// TwinCAT 3 PLC project Hboy
// ProgramVersion: 3.1.4023.0
// libraries:
//   Tc2_MC2, * (Beckhoff Automation GmbH)
//   Tc2_Standard, * (Beckhoff Automation GmbH)
//   Tc2_System, * (Beckhoff Automation GmbH)
//   Tc2_SystemCX, * (Beckhoff Automation GmbH)
//   Tc2_Utilities, * (Beckhoff Automation GmbH)
//   Tc3_Module, * (Beckhoff Automation GmbH)
//   XboxControllerUtilities, * (Beckhoff Community)
// project tree:
//   DUTs/ Controller.TcDUT, Pos.TcDUT
//   GVLs/ GVL.TcGVL
//   / PlcTask.TcTTO
//   POUs/ E_Stop.TcPOU, HbotForwardKinematics.TcPOU, LimitSwitches.TcPOU, TcXbox.TcPOU, MovementTypeSelector.TcPOU, PrepareAxes.TcPOU, MAIN.TcPOU
//   POUs/MovementType_Gcode/ FB_Movement_Gcode.TcPOU, FB_GcodeAgent.TcPOU
//   POUs/MovementType_Teach/ FB_Frames.TcPOU, FB_Movement_Teach.TcPOU, FB_Movement_Xbox.TcPOU, Frame.TcDUT
//   POUs/Hbot_Kinematics/ FB_HbotHome.TcPOU, FB_HbotKinematics.TcPOU, FB_HbotMovement.TcPOU, FB_PowerAll.TcPOU, FB_ResetAll.TcPOU
// real-time tasks:
//   TASK PlcTask: cycle T#1ms, priority 20, ADS port 350
//   TASK Job Task: cycle default, priority 32
// motion (NC):
//   TASK NC-Task 1 SAF: cycle T#2ms, priority 4, ADS port 501
//   TASK NC-Task 1 SVB: cycle T#10ms, priority 8, ADS port 511
//   AXIS Axis A (id 1)
//     Dynamic: Acceleration=20631.2, Deceleration=20631.2, Jerk=1237870, DelayTime=0.008
//     Velo: RefSearch=6.87706, RefSync=6.87706, SlowManual=150, FastManual=200, Fast=2347.941, Maximum=687.706
//     OtherSettings: AllowMotionCmdToSlave=true
//     encoder EncType=19
//       EncPara: ScaleFactorNumerator=60, ScaleFactorDenominator=1048576, MaxCount=#xffffffff
//     drive DrvType=16
//       DrvPara: MaxCount=#xffffffff, DriveControlDWord=#x00020100
//         Analog: VeloReferenz=756.4766, TorqueSetpointScale=10, ScaleFactorActTorque=0.1
//         TimeComp: TaskDelayCycles=1
//     controller CtrType=1
//       CtrPara: PriorControlFactor=1
//         PosDiffControl: Enable=false
//         Observer: BandWidth=20
//   AXIS Axis B (id 2)
//     Dynamic: Acceleration=15768.4, Deceleration=15768.4, Jerk=2468790, DelayTime=0.008
//     Velo: RefSearch=6.87706, RefSync=6.87706, SlowManual=150, FastManual=200, Fast=687.706, Maximum=687.706
//     OtherSettings: AllowMotionCmdToSlave=true
//     encoder EncType=19
//       EncPara: ScaleFactorNumerator=60, ScaleFactorDenominator=1048576, Inverse=true, MaxCount=#xffffffff
//     drive DrvType=16
//       DrvPara: Inverse=true, MaxCount=#xffffffff, DriveControlDWord=#x00020100
//         Analog: VeloReferenz=756.4766, TorqueSetpointScale=10, ScaleFactorActTorque=0.1
//         TimeComp: TaskDelayCycles=1
//     controller CtrType=1
//       CtrPara: PriorControlFactor=1
//         PosDiffControl: Enable=false
//         Observer: BandWidth=20
// I/O:
//   DEVICE Device 1 (EtherCAT), AmsNetId 5.71.241.84.2.1
//     Term 1 (EK1200) [EK1200-5000 EtherCAT Power supply (2A E-Bus)]
//       Term 8 (EL1012) [EL1012 2Ch. Dig. Input 24V, 10µs]
//       Term 2 (EL6900) [EL6900, TwinSAFE PLC]
//       Term 3 (EL1904) [EL1904, 4 Ch. Safety Input 24V, TwinSAFE]
//         modules: Module 1 (FSOES)
//       Term 4 (EL2904) [EL2904, 4 Ch. Safety Output 24V, 0.5A, TwinSAFE]
//         modules: Module 1 (FSOES), Module 2 (DO)
//       Term 5 (ELM7222-0010) [ELM7222-0010 2Ch. Servo Terminal (48 V, 8 A RMS, OCT)]
//       Term 6 (EL1088) [EL1088 8Ch. Dig. Input 24V, 3ms, negative]
//       Term 7 (EL9011) [EL9011 End Terminal]
//   DEVICE Device 5 (USB)
//     Box 1 (CX2100 Power Supply)
// variable links:
//   Device 1 (EtherCAT) <-> Device 1 (EtherCAT)/Term 1 (EK1200)/Term 2 (EL6900)
//     Term 1 (EK1200)/Term 3 (EL1904)/Module 1 (FSOES)/RxPDO/FSOE <-> ConnectionInputs/Message_9 TxPDO
//     Term 1 (EK1200)/Term 4 (EL2904)/Module 1 (FSOES)/RxPDO/FSOE <-> ConnectionInputs/Message_10 TxPDO
//     Term 1 (EK1200)/Term 3 (EL1904)/Module 1 (FSOES)/TxPDO/FSOE <-> ConnectionOutputs/Message_9 RxPDO
//   Device 1 (EtherCAT) <-> Device 1 (EtherCAT)/Term 1 (EK1200)/Term 4 (EL2904)
//     Term 1 (EK1200)/Term 2 (EL6900)/ConnectionOutputs/Message_10 RxPDO <-> Module 1 (FSOES)/TxPDO/FSOE
//   NC-Task 1 SAF/Axes/Axis A <-> Device 1 (EtherCAT)/Term 1 (EK1200)/Term 5 (ELM7222-0010)
//     Drive/Inputs/In/nDataIn1 <-> DRV Following error actual value Channel 1/Following error actual value
//     Drive/Inputs/In/nDcOutputTime <-> InfoData/DcOutputShift
//     Drive/Inputs/In/nState1 <-> DRV Statusword Channel 1/Statusword
//     Drive/Inputs/In/nState2 <-> DRV Statusword Channel 1/Statusword @bit 8
//     Drive/Inputs/In/nState4 @bit 1 <-> WcState/InputToggle
//     Drive/Inputs/In/nState4 <-> WcState/WcState
//     Drive/Outputs/Out/nCtrl1 <-> DRV Controlword Channel 1/Controlword
//     Drive/Outputs/Out/nCtrl2 <-> DRV Controlword Channel 1/Controlword @bit 8
//     Drive/Outputs/Out/nDataOut1 <-> DRV Target position Channel 1/Target position
//     Enc/Inputs/In/nDataIn1 <-> FB Position Channel 1/Position
//     Enc/Inputs/In/nDcInputTime <-> InfoData/DcInputShift
//     Enc/Inputs/In/nState4 @bit 1 <-> WcState/InputToggle
//     Enc/Inputs/In/nState4 <-> WcState/WcState
//   NC-Task 1 SAF/Axes/Axis B <-> Device 1 (EtherCAT)/Term 1 (EK1200)/Term 5 (ELM7222-0010)
//     Drive/Inputs/In/nDataIn1 <-> DRV Following error actual value Channel 2/Following error actual value
//     Drive/Inputs/In/nDcOutputTime <-> InfoData/DcOutputShift
//     Drive/Inputs/In/nState1 <-> DRV Statusword Channel 2/Statusword
//     Drive/Inputs/In/nState2 <-> DRV Statusword Channel 2/Statusword @bit 8
//     Drive/Inputs/In/nState4 @bit 1 <-> WcState/InputToggle
//     Drive/Inputs/In/nState4 <-> WcState/WcState
//     Drive/Outputs/Out/nCtrl1 <-> DRV Controlword Channel 2/Controlword
//     Drive/Outputs/Out/nCtrl2 <-> DRV Controlword Channel 2/Controlword @bit 8
//     Drive/Outputs/Out/nDataOut1 <-> DRV Target position Channel 2/Target position
//     Enc/Inputs/In/nDataIn1 <-> FB Position Channel 2/Position
//     Enc/Inputs/In/nDcInputTime <-> InfoData/DcInputShift
//     Enc/Inputs/In/nState4 @bit 1 <-> WcState/InputToggle
//     Enc/Inputs/In/nState4 <-> WcState/WcState
//   Hboy/Hboy Instance <-> Device 1 (EtherCAT)/Term 1 (EK1200)/Term 2 (EL6900)
//     PlcTask Inputs/E_Stop.UserEStopButton <-> StandardInputs/Standard Out Var 8
//     PlcTask Inputs/E_Stop.UserResetButton <-> StandardInputs/Standard Out Var 11
//     PlcTask Outputs/GVL.SafetyErrAck <-> StandardOutputs/Standard In Var 1
//     PlcTask Outputs/GVL.SafetyRun <-> StandardOutputs/Standard In Var 2
//   Hboy/Hboy Instance <-> Device 1 (EtherCAT)/Term 1 (EK1200)/Term 6 (EL1088)
//     PlcTask Inputs/MovementTypeSelector.fbXbox.leftSwitch <-> Channel 4/Input
//     PlcTask Inputs/MovementTypeSelector.fbXbox.rightSwitch <-> Channel 2/Input
//   Hboy/Hboy Instance <-> Device 1 (EtherCAT)/Term 1 (EK1200)/Term 8 (EL1012)
//     PlcTask Inputs/MovementTypeSelector.fbXbox.balluff_neg <-> Channel 2/Input
//     PlcTask Inputs/MovementTypeSelector.fbXbox.balluff_pos <-> Channel 1/Input
//   Hboy/Hboy Instance <-> NC-Task 1 SAF/Axes/Axis A
//     PlcTask Inputs/GVL.StepperReferenceA.NcToPlc <-> Outputs/ToPlc
//     PlcTask Outputs/GVL.StepperReferenceA.PlcToNc <-> Inputs/FromPlc
//   Hboy/Hboy Instance <-> NC-Task 1 SAF/Axes/Axis B
//     PlcTask Inputs/GVL.StepperReferenceB.NcToPlc <-> Outputs/ToPlc
//     PlcTask Outputs/GVL.StepperReferenceB.PlcToNc <-> Inputs/FromPlc

CONFIGURATION Hboy
    RESOURCE PLC ON TwinCAT3
        TASK PlcTask(INTERVAL := T#1ms, PRIORITY := 20);
        PROGRAM MAIN WITH PlcTask : MAIN;
        PROGRAM HbotForwardKinematics WITH PlcTask : HbotForwardKinematics;
    END_RESOURCE
END_CONFIGURATION

// ---- DUTs/Controller.TcDUT
TYPE Controller :
STRUCT
	bDpadRight : BOOL;
	bDpadLeft : BOOL;
	bDpadUp : BOOL;
	bDpadDown : BOOL;
	bAbtn : BOOL;
	bBbtn : BOOL;
	bXbtn : BOOL;
	bYbtn : BOOL;
	rightStick : ARRAY[0..2] OF REAL;
	leftStick : ARRAY[0..2] OF REAL;
END_STRUCT
END_TYPE

// ---- DUTs/Pos.TcDUT
TYPE Pos :
STRUCT
	x : REAL;
	y : REAL;
END_STRUCT
END_TYPE

// ---- POUs/MovementType_Teach/Frame.TcDUT
TYPE Frame :
STRUCT
	Name : STRING;
	X : REAL;
	Y : REAL;
END_STRUCT
END_TYPE

// ---- GVLs/GVL.TcGVL
{attribute 'qualified_only'}
VAR_GLOBAL
	StepperReferenceA	:	AXIS_REF;
	StepperReferenceB	:	AXIS_REF;
	LimitSwitchMidLeft 		AT %I* : 	BOOL;
	LimitSwitchMidRight 	AT %I* : 	BOOL;
	LimitSwitchBotLeft		AT %I* : 	BOOL;
	LimitSwitchBotRight 	AT %I* :	BOOL;
	LimitSwitchTopLeft		AT %I* : 	BOOL;
	LimitSwitchTopRight		AT %I* : 	BOOL;	
	SafetyRun         AT %Q*      :   BOOL;
	SafetyReset       AT %Q*      :   BOOL;
	SafetyErrAck      AT %Q*      :   BOOL;
END_VAR

// ---- POUs/MAIN.TcPOU
PROGRAM MAIN
VAR
	start: BOOL;
	caseswitch: (prepare, starting, selectmovement);
	lool : T_AmsNetID := 'asdasd';
	ProcessXbox: NT_StartProcess;
	idk : UINT; 	
	displayTest : FB_CXSetTextDisplayUSB := (bExecute := TRUE);
END_VAR

//PrepareAxes();
//HbotForwardKinematics();
//nig(CLK := yee);
//gcodeagent(bExecute := TRUE, bNextLine := yee);
//IF PrepareAxes.switchcase = PrepareAxes.movement THEN
//	;
//END_IF

displayTest(
	bExecute:= , 
	sNetID:= , 
	nPort:= 28928, 
	eMode:= eCX2100_WriteLines, 
	sLine1:= '   Welcome to   ', 
	sLine2:= '   ITAP 2023!   ', 
	nCursorPosX:= , 
	nCursorPosY:= , 
	bBusy=> , 
	bError=> , 
	nErrorID=> );

TcXbox();

//GVL.LimitSwitchX := TcXbox.xBoxController.P_Buttons.bA_Button;
//GVL.LimitSwitchY := TcXbox.xBoxController.P_Buttons.bB_Button;

start := tcXbox.xBoxController.P_Buttons.bStart; //addded 20230711 to avoid the need to use HMI to initialise

CASE caseswitch OF
	starting:
		IF start THEN
			caseswitch := Prepare;
		END_IF
		
	Prepare: 
	PrepareAxes();
	IF PrepareAxes.bDone THEN
		caseswitch := selectmovement;
	END_IF
	
	selectmovement:
		MovementTypeSelector();
		GVL.SafetyRun := TRUE;
		
END_CASE

E_Stop();
LimitSwitches();
//C:\Users\weikoons.BECKHOFF\Downloads\HBot_SelfDefinedKinematics\HBot_SelfDefinedKinematics\Hboy\POUs\MovementType_Teach

//ProcessXbox(PATHSTR := 'C:\Users\MaxwellA.BECKHOFF\Documents\TcXaeShell\HBot_SelfDefinedKinematics\HBot_SelfDefinedKinematics\Hboy\POUs\MovementType_Teach\xboxcontrol.exe', 
					//	DIRNAME := 'C:\Users\MaxwellA.BECKHOFF\Documents\TcXaeShell\HBot_SelfDefinedKinematics\HBot_SelfDefinedKinematics\Hboy\POUs\MovementType_Teach\',
						//COMNDLINE := 'GVL.controller 127.0.0.1.1.1',
						//START := TRUE);

END_PROGRAM

// ---- POUs/TcXbox.TcPOU
PROGRAM TcXbox
VAR
	xBoxController : FB_XBOX_Controller(NETID := '', iControllerNumber := 1);
	
	StartXbox : NT_StartProcess;
	
	bIsconnected : BOOL;
	
	t1 : TIME := T#10M;
	t2 : TIME := T#2S;
	t3 : TIME;
	t4 : UDINT;
	
	arrTest : ARRAY [0..9] OF BOOL;
	
END_VAR

StartXbox(
	NETID:= , 
	PATHSTR:= 'C:\Program Files\Beckhoff Community\TwinCAT Xbox Controller Service\ADS-Controller-Server.exe', 
	DIRNAME:= 'C:\Program Files\Beckhoff Community\TwinCAT Xbox Controller Service', 
	COMNDLINE:= , 
	START:= TRUE, 
	TMOUT:= , 
	BUSY=> , 
	ERR=> , 
	ERRID=> );

xBoxController.Cycle();

bIsconnected := xboxController.P_Status.bConnected;

END_PROGRAM

// ---- POUs/PrepareAxes.TcPOU
PROGRAM PrepareAxes
VAR
	switchcase : (Chilling, Reset, Power, Movement, lol, Error);
	limitx : BOOL;
	limity : BOOL;
	
	// define kinematics objects
	fbBot : FB_HbotMovement;
	fbHome : FB_HbotHome;
	X : REAL;
	Y : REAL;
	mode : STRING;
	yee : BOOL;
	rere : ARRAY[0..1] OF REAL;
	
	// grouped fb
	fbResetAll : FB_ResetAll;
	fbPowerAll : FB_PowerAll;
	
	// done indicator
	bDone : BOOL;
	bError : BOOL;
END_VAR

CASE switchcase OF
	Chilling:
		fbResetAll(io_M1 := GVL.StepperReferenceA, io_M2 := GVL.StepperReferenceB, bExecute := FALSE);
		switchcase := Reset;
		
	Reset:
		fbResetAll(io_M1 := GVL.StepperReferenceA, io_M2 := GVL.StepperReferenceB, bExecute := TRUE);
		IF fbResetAll.bDone THEN
			switchcase := Power;
		ELSIF fbResetAll.bError THEN
			switchcase := Error;
		END_IF
		
	Power:
		fbPowerAll(bEnable := TRUE, io_M1 := GVL.StepperReferenceA, io_M2 := GVL.StepperReferenceB);
		IF fbPowerAll.bStatus THEN
			switchcase := Movement;
		ELSIF fbPowerAll.bError THEN
			switchcase := Error;
		END_IF
	Movement:
		bDone := TRUE;
//		fbBot(MovementMode:= fbBot.MoveRelative, rDeltaX:= X, rDeltaY := Y, bExecute := yee,
//				StepperA := GVL.StepperReferenceA, StepperB := GVL.StepperReferenceB, rLinearSpeed := 100,
//				rCurrentX := HbotForwardKinematics.rCurrentX, rCurrentY := HbotForwardKinematics.rCurrentY);
//		fbHome(bExecute := yee, Velocity := 100, StepperA := GVL.StepperReferenceA, StepperB := GVL.StepperReferenceB, limitSwitchX := limitx, limitSwitchY  := limity);
//		IF fbBot.bDone THEN
//			switchcase := lol;
//		END_IF
//		IF fbBot.bError THEN
//			switchcase := Error;
//		END_IF
		;
	Error:
		bError := TRUE;
		switchcase := Chilling;
END_CASE

END_PROGRAM

// ---- POUs/Hbot_Kinematics/FB_HbotMovement.TcPOU
FUNCTION_BLOCK FB_HbotMovement EXTENDS FB_HbotKinematics
VAR_INPUT
	MovementMode : INT := MoveAbsolute;
	rLinearSpeed : REAL;
	rCurrentX : REAL;
	rCurrentY : REAL;
	rDeltaX : REAL;
	rDeltaY : REAL;
	bExecute : BOOL;
	rTarget : ARRAY[0..1] OF REAL;
END_VAR
VAR_OUTPUT
	bDone : BOOL;
	bError : BOOL;
	bBusy : BOOL;
END_VAR
VAR
	McMoveAbsA : MC_MoveAbsolute;
	McMoveAbsB : MC_MoveAbsolute;
	McMoveRelA : MC_MoveRelative;
	McMoveRelB : MC_MoveRelative;
	
	aRotationalDisplacement : ARRAY [0..1] OF REAL;
	aRotationalVelocity : ARRAY [0..1] OF REAL;
	bBypass: ARRAY[0..1] OF BOOL;
	
	MoveRelative : INT := 1;
	MoveAbsolute : INT := 0;
END_VAR
VAR_IN_OUT
	StepperA	:	AXIS_REF;
	StepperB	:	AXIS_REF;
END_VAR

IF McMoveAbsA.Error OR McMoveAbsB.Error OR McMoveRelA.Error OR McMoveRelB.Error THEN
	bError := TRUE;
END_IF

IF bExecute AND NOT bError THEN
	bDone := FALSE;
	IF MovementMode = MoveAbsolute THEN
		rTarget[0] := rDeltaX - rCurrentX;
		rTarget[1] := rDeltaY - rCurrentY;
		aRotationalDisplacement := CalculateAxisRotationRelative(rDeltaX, rDeltaY); // calculate displacement
		aRotationalVelocity := CalculateVelocities(rTarget[0], rTarget[1], rLinearSpeed); // calculate velocity
	ELSE
		rTarget[0] := rDeltaX;
		rTarget[1] := rDeltaY;
		aRotationalDisplacement := CalculateAxisRotationRelative(rTarget[0], rTarget[1]); // calculate displacement
		aRotationalVelocity := CalculateVelocities(rTarget[0], rTarget[1], rLinearSpeed); // calculate velocity
	END_IF
	
	// checking if displacement or velocity is 0, if so, don't move the stepper
	IF aRotationalVelocity[0] = 0 THEN
		bBypass[0] := TRUE;
	END_IF
	
	IF aRotationalVelocity[1] = 0 THEN
		bBypass[1] := TRUE;
	END_IF
	
	//===================== checking if the movement is absolute or relative=======================
	IF MovementMode = MoveRelative THEN
		IF NOT bBypass[0] THEN // check edge case
			McMoveRelA(Axis := StepperA, Execute := TRUE, Distance := aRotationalDisplacement[0], Velocity := aRotationalVelocity[0]);
		END_IF
		
		IF NOT bBypass[1] THEN // check edge case
			McMoveRelB(Axis := StepperB, Execute := TRUE, Distance := aRotationalDisplacement[1], Velocity := aRotationalVelocity[1]);
		END_IF
		bBusy := TRUE;
		
		IF (McMoveRelA.Done OR bBypass[0]) AND (McMoveRelB.Done OR bBypass[1]) THEN
			bBusy := FALSE;
			bDone := TRUE;
			McMoveRelA(Axis := StepperA, Execute := FALSE);
			McMoveRelB(Axis := StepperB, Execute := FALSE);
			bExecute := FALSE;
			bBypass[0] := FALSE;
			bBypass[1] := FALSE;
		END_IF
	
	ELSIF MovementMode = MoveAbsolute THEN
		IF NOT bBypass[0] THEN
			McMoveAbsA(Axis := StepperA, Execute := TRUE, Position := aRotationalDisplacement[0], Velocity := aRotationalVelocity[0]);
		END_IF
		
		IF NOT bBypass[1] THEN
			McMoveAbsB(Axis := StepperB, Execute := TRUE, Position := aRotationalDisplacement[1], Velocity := aRotationalVelocity[1]);
		END_IF
		bBusy := TRUE;
		
		IF (McMoveAbsA.Done OR bBypass[0]) AND (McMoveAbsB.Done OR bBypass[1]) THEN
			bBusy := FALSE;
			bDone := TRUE;
			McMoveAbsA(Axis := StepperA, Execute := FALSE);
			McMoveAbsB(Axis := StepperB, Execute := FALSE);
			bExecute := FALSE;
			bBypass[0] := FALSE;
			bBypass[1] := FALSE;
		END_IF
	END_IF
END_IF

END_FUNCTION_BLOCK

// ---- POUs/Hbot_Kinematics/FB_HbotKinematics.TcPOU
FUNCTION_BLOCK FB_HbotKinematics
VAR_INPUT
END_VAR
VAR_OUTPUT
END_VAR
VAR
END_VAR

METHOD CalculateAxisRotationRelative : ARRAY[0..1] OF REAL; // returns [a,b]
VAR_INPUT
	rDeltaX : REAL;
	rDeltaY : REAL;
END_VAR
VAR
	returnableArray : ARRAY[0..1] OF REAL;
	polar : ARRAY[0..1] OF REAL;
END_VAR
//polar := PolarCoordinates(DeltaX := rDeltaX, DeltaY := rDeltaY);
returnableArray[0] := -rDeltaX - rDeltaY;
returnableArray[1] := -rDeltaX + rDeltaY;
CalculateAxisRotationRelative := returnableArray;
END_METHOD

METHOD CalculateVelocities : ARRAY[0..1] OF REAL
VAR_INPUT
	rDeltaX : REAL;
	rDeltaY : REAL;
	rLinearSpeed : REAL;
END_VAR
VAR
	returnableArray : ARRAY[0..1] OF REAL;
	rAngle : REAL;
END_VAR
rAngle := GetAngleFromXY(rDeltaX := rDeltaX, rDeltaY := rDeltaY);
returnableArray[0] := ABS(rLinearSpeed * COS(rAngle) + rLinearSpeed * SIN(rAngle));
returnableArray[1] := ABS(rLinearSpeed * COS(rAngle) - rLinearSpeed * SIN(rAngle));
CalculateVelocities := returnableArray;
END_METHOD

METHOD GetAngleFromXY : REAL
VAR_INPUT
	rDeltaX : REAL;
	rDeltaY : REAL;
END_VAR
IF rDeltaX = 0 THEN
	rDeltaX := 0.0000001;
END_IF
IF rDeltaY = 0 THEN
	rDeltaY := 0.0000001;
END_IF
GetAngleFromXY := ATAN(rDeltaX/rDeltaY);
END_METHOD

END_FUNCTION_BLOCK

// ---- POUs/Hbot_Kinematics/FB_HbotHome.TcPOU
FUNCTION_BLOCK FB_HbotHome
VAR_INPUT
	bExecute : BOOL;
	Velocity : REAL;
END_VAR
VAR_OUTPUT
	bDone : BOOL;
	bError : BOOL;
	bBusy : BOOL;
END_VAR
VAR
	init : R_TRIG;
	StepperAJog : MC_Jog;
	StepperBJog : MC_Jog;
	
	StepperASetPos : MC_SetPosition;
	StepperBSetPos : MC_SetPosition;
	
	StepperAHome : MC_Home;
	StepperBHome : MC_Home;
	
	StepperAHalt : MC_Halt;
	StepperBHalt : MC_Halt;
	
	homeSequence : (homeX, homeY, halt, forcecalibration, done, error);
	ErrorTimeout : ton;
	ErrorTimeoutCase : INT;
END_VAR
VAR_IN_OUT
	StepperA	:	AXIS_REF;
	StepperB	:	AXIS_REF;
	
	limitSwitchX : BOOL;
	limitSwitchY : BOOL;
END_VAR

init(CLK := bExecute); // detect rising edge

IF bExecute AND NOT bError THEN 
	IF init.Q THEN // if it is on rising edge (i.e, first instance of bexecute is true
		homeSequence := homeX; // set switch case to homeX
	END_IF
	
	CASE homeSequence OF
	homeX :
		bBusy := TRUE;
		bDone := FALSE;
		// Home Cartesian X, Both steppers to jog forward at the same speed
		StepperAJog(Axis := StepperA, JogForward := TRUE, Velocity := Velocity);
		StepperBJog(Axis := StepperB, JogForward := TRUE, Velocity := Velocity);
		IF StepperAJog.Error OR StepperBJog.Error THEN
			homeSequence := error;
		END_IF
		IF limitSwitchX THEN // if limit switch is triggered, stop jogging and go to homeY case
			StepperAJog(Axis := StepperA, JogForward := FALSE);
			StepperBJog(Axis := StepperB, JogForward := FALSE);
			homeSequence := homeY;
		END_IF
		IF StepperAJog.CommandAborted OR StepperBJog.CommandAborted THEN 
			homeSequence := Error;
		END_IF
	
	homeY :
		// Home Cartesian Y, Both steppers to jog in opposite directions at the same speed
		StepperAJog(Axis := StepperA, JogForward := TRUE, Velocity := Velocity);
		StepperBJog(Axis := StepperB, JogBackwards := TRUE, Velocity := Velocity);
		IF StepperAJog.Error OR StepperBJog.Error THEN
			homeSequence := error;
		END_IF
		IF limitSwitchY THEN // if limit switch is triggered, stop jogging and go to halt case
			StepperAJog(Axis := StepperA, JogForward := FALSE);
			StepperBJog(Axis := StepperB, JogBackwards := FALSE);
			homeSequence := halt;
		END_IF
		
		IF StepperAJog.CommandAborted OR StepperBJog.CommandAborted THEN 
			homeSequence := Error;
		END_IF
		
	halt :
		// halting motors
		StepperAHalt(Axis := StepperA, Execute := TRUE);
		StepperBHalt(Axis := StepperB, Execute := TRUE);
		IF StepperAHalt.Done AND StepperBHalt.Done THEN
			homeSequence := forcecalibration; // once stopped, reset mc_halt and go to force calibration case
			StepperAHalt(Axis := StepperA, Execute := FALSE);
			StepperBHalt(Axis := StepperB, Execute := FALSE);
		ELSIF StepperAHalt.Error OR StepperBHalt.Error THEN
			homeSequence := error;
		END_IF
		
		
	forcecalibration :
		// set stepper positions to 0
		StepperASetPos(Axis := StepperA, Position := 0.0, Mode := FALSE, Execute := TRUE);
		StepperBSetPos(Axis := StepperB, Position := 0.0, Mode := FALSE, Execute := TRUE);
		IF StepperASetPos.Error OR StepperBSetPos.Error THEN
			homeSequence := error;
		ELSIF StepperASetPos.Done AND StepperBSetPos.Done THEN
			homeSequence := done; // go to done case
			StepperASetPos(Axis := StepperA, Position := 0.0, Mode := FALSE, Execute := FALSE);
			StepperBSetPos(Axis := StepperB, Position := 0.0, Mode := FALSE, Execute := FALSE);
		END_IF
		
	done :
		bDone := TRUE;
		bBusy := FALSE;
		
	error:
	
		CASE ErrorTimeoutCase OF 
		0: bError := TRUE;
		ErrorTimeout (IN := TRUE, PT := T#5000MS);
		IF ErrorTimeout.Q THEN 
			ErrorTimeoutCase := 10; 
		END_IF
		10: bError := FALSE; 
		homeSequence := done;
		ErrorTimeoutCase := 0; 
		
		END_CASE
		
	END_CASE
ELSE
	bDone := FALSE;
END_IF

END_FUNCTION_BLOCK

// ---- POUs/Hbot_Kinematics/FB_ResetAll.TcPOU
FUNCTION_BLOCK FB_ResetAll
VAR_INPUT
	bExecute : BOOL;
END_VAR
VAR_OUTPUT
	bDone : BOOL;
	bError : BOOL;
END_VAR
VAR
	reset1 : MC_Reset;
	reset2 : MC_Reset;
END_VAR
VAR_IN_OUT
	io_M1 : AXIS_REF;
	io_M2 : AXIS_REF;
END_VAR

reset1(Axis := io_M1, Execute := bExecute);
reset2(Axis := io_M2, Execute := bExecute);

bError := reset1.Error OR reset2.Error;
bDone := reset1.Done AND reset2.Done AND NOT bError;

END_FUNCTION_BLOCK

// ---- POUs/Hbot_Kinematics/FB_PowerAll.TcPOU
FUNCTION_BLOCK FB_PowerAll
VAR_INPUT
	bEnable : BOOL;
END_VAR
VAR_OUTPUT
	bStatus : BOOL;
	bError : BOOL;
END_VAR
VAR
	power1 : MC_Power;
	power2 : MC_Power;
END_VAR
VAR_IN_OUT
	io_M1 : AXIS_REF;
	io_M2 : AXIS_REF;
END_VAR

power1(Axis := io_M1, Enable := bEnable, Enable_Negative := bEnable, Enable_Positive := bEnable);
power2(Axis := io_M2, Enable := bEnable, Enable_Negative := bEnable, Enable_Positive := bEnable);

bError := power1.Error OR power2.Error;
bStatus := power1.Status AND power2.Status AND NOT bError;

END_FUNCTION_BLOCK

// ---- POUs/MovementTypeSelector.TcPOU
PROGRAM MovementTypeSelector
VAR
	fbGcode : FB_Movement_Gcode;
	fbHome : FB_HbotHome;
	fbXbox : FB_Movement_Xbox;
	limx : BOOL;
	limy : BOOL;
	
	caseswitch : (none, home, gcode, teach, vision, error);
END_VAR

CASE caseswitch OF
	none:
	fbGcode(bExecute := FALSE);
	fbXbox(bExecute := FALSE);
	fbHome(bExecute := FALSE, StepperA := GVL.StepperReferenceA, StepperB := GVL.StepperReferenceB,limitSwitchX := GVL.LimitSwitchMidLeft, limitSwitchY := GVL.LimitSwitchBotLeft);
		(* 20230712: Decoupling from HMI, for now clicking on Xbox Controller's Select btn goes to Teach *)
		IF tcXbox.xBoxController.P_Buttons.bB_Button THEN
			caseswitch := teach;
		END_IF
		
		(* Home first before going into Teach If you do not, it will take its current location as "0" although it technically doesnt matter for now*)
		(*IF TcXbox.xBoxController.P_Buttons.bA_Button THEN 
			caseswitch := home;
		END_IF*) //UNCOMMENT AFTER LIMIT SWITCHES ARE READY YOU RETARD 
		
	home:
		fbHome(bExecute := TRUE, StepperA := GVL.StepperReferenceA, StepperB := GVL.StepperReferenceB,
			limitSwitchX := GVL.LimitSwitchMidLeft, limitSwitchY := GVL.LimitSwitchBotLeft);
		IF fbHome.bError THEN
			caseswitch := error;
		ELSIF fbHome.bDone THEN
			fbHome(bExecute := FALSE, StepperA := GVL.StepperReferenceA, StepperB := GVL.StepperReferenceB,
			limitSwitchX := GVL.LimitSwitchMidLeft, limitSwitchY := GVL.LimitSwitchBotLeft);
			caseswitch := none;
		END_IF
		
	gcode:
		fbGcode(bExecute := TRUE);
		IF fbGcode.bFinished AND NOT fbGcode.initial.Q THEN
			caseswitch := none;
		END_IF
		
	teach:
		fbXbox(bExecute := TRUE);

	Error:
		caseswitch := None;
		
END_CASE

END_PROGRAM

// ---- POUs/MovementType_Gcode/FB_Movement_Gcode.TcPOU
FUNCTION_BLOCK FB_Movement_Gcode
VAR_INPUT
	bExecute : BOOL;
END_VAR
VAR_OUTPUT
	bBusy : BOOL;
	bError : BOOL;
	bFinished : BOOL;
	initial : R_TRIG;
END_VAR
VAR
	gcodeagent : FB_GcodeAgent;
	// define kinematics objects
	fbMover : FB_HbotMovement;
	fbHome : FB_HbotHome;
	sGodeFileName : STRING;
	caseswitch : (init, prep, movement, end, error);
END_VAR

initial(CLK := bExecute);
IF initial.Q THEN // on initial trigger, run initilsation case to initiate gcode and reset variables
	caseswitch := init;
	bFinished := FALSE;
	bBusy := TRUE;
	gcodeagent.bEnd := FALSE;
END_IF
CASE caseswitch OF
	init:
		IF sGodeFileName <> '' THEN
			IF bExecute AND NOT bError THEN
			gcodeagent(sGcodeFile := sGodeFileName, sFBName := 'MovementTypeSelector.fbGcode.gcodeagent', bExecute := bExecute);
			// run gcode agent python script
			IF NOT gcodeagent.Process.BUSY THEN 
				caseswitch := prep;
			END_IF
		END_IF
		END_IF
	prep:
		fbMover( bExecute := FALSE, StepperA := GVL.StepperReferenceA, StepperB := GVL.StepperReferenceB); // stop all movement
		IF gcodeagent.bWriteDone THEN // wait for gcode agent to write a new line before going to next step
			caseswitch := movement;
		END_IF
		IF gcodeagent.bEnd THEN
			caseswitch := end; // if gcode agent sends a end command, go to end case
		END_IF
	movement:
		fbMover(MovementMode := fbMover.MoveAbsolute,
				rLinearSpeed := 60,
				rCurrentX := HbotForwardKinematics.rCurrentX,
				rCurrentY := HbotForwardKinematics.rCurrentY,
				rDeltaX := gcodeagent.x,
				rDeltaY := gcodeagent.y,
				bExecute := TRUE,
				StepperA := GVL.StepperReferenceA,
				StepperB := GVL.StepperReferenceB); // once gcode is received, move to positions
				 
		IF fbMover.bError THEN
			caseswitch := error; //catch errors
		ELSIF fbMover.bDone THEN
			caseswitch := prep; // if it is done, go to the prep switch case
			gcodeagent.bNextLine := TRUE; // send signal to python script to show that the movement is completed
		END_IF
	end:
		bFinished := TRUE;
		bBusy := FALSE;
		gcodeagent(sGcodeFile := 'choppt.gcode', sFBName := 'MovementTypeSelector.fbGcode.gcodeagent', bExecute := FALSE);
	error:
		bError := TRUE;
END_CASE

END_FUNCTION_BLOCK

// ---- POUs/MovementType_Gcode/FB_GcodeAgent.TcPOU
FUNCTION_BLOCK FB_GcodeAgent
VAR_INPUT
	bExecute : BOOL;
	bNextLine : BOOL;
	bWriteDone : BOOL;
	sGcodeFile : STRING;
	sFBName : STRING;
	bEnd : BOOL;
END_VAR
VAR_OUTPUT
	x : REAL;
	y : REAL;
	z : REAL;
	e : REAL;
	f : REAL;
END_VAR
VAR
	trig : R_TRIG;
	Process : NT_StartProcess;
	sCommand : STRING(1000);
	placeholder : ARRAY [0..200] OF STRING(200);
END_VAR
//'main.py choppt.gcode MovementTypeSelector.fbGcode.gcodeagent 10.123.67.6.1.1'

// prepare command to run python script]
trig(CLK := bExecute);
placeholder[0] := sGcodeFile;
placeholder[1] := ' ';
placeholder[2] := sFBName;
placeholder[3] := ' ';
placeholder[4] := HbotForwardKinematics.fbAms.AddrString;

sCommand := ConcatAll(placeholder); //concat all

Process(NETID := '10.123.6.66.1.1',
		COMNDLINE := sCommand,
		PATHSTR := 'C:\Users\weikoons.BECKHOFF\Downloads\HBot_SelfDefinedKinematics\HBot_SelfDefinedKinematics\Hboy\POUs\MovementType_Gcode\main.exe',
//		DIRNAME := 'C:\Users\MaxwellA.BECKHOFF\Desktop\Coding\Python\asd\Gcode',
		START := trig.Q); // start process

METHOD ConcatAll : STRING(1000)
VAR_INPUT
	allString : ARRAY [0..200] OF STRING(200);
END_VAR
VAR
	resultString : STRING(1000);
	i : INT;
END_VAR
FOR i := 0 TO 199 DO
	IF allString[i] = '' THEN
		ConcatAll := resultString;
	END_IF
	resultString := CONCAT(resultString, allString[i]);
END_FOR
ConcatAll := resultString;
END_METHOD

END_FUNCTION_BLOCK

// ---- POUs/HbotForwardKinematics.TcPOU
PROGRAM HbotForwardKinematics
VAR
	rCurrentY : REAL;
	rCurrentX : REAL;
	
	HMIX : REAL;
	HMIY : REAL;
	
	currentpos : Pos;
	len : ULINT := 4000;
	hist : ARRAY[1..1, 0..4000] OF Pos;
	i : ULINT;
	timer : TON;
	fbAms : FB_GetLocalAmsNetId;
	bReqStarted : BOOL := TRUE;
END_VAR

// calculating real time positions based on axes A and B
rCurrentX := (-GVL.StepperReferenceA.NcToPlc.ActPos - GVL.StepperReferenceB.NcToPlc.ActPos)/2;
rCurrentY := (-GVL.StepperReferenceA.NcToPlc.ActPos + GVL.StepperReferenceB.NcToPlc.ActPos)/2;
HMIX := Round2dp(rCurrentX);
HMIY := Round2dp(rCurrentY);

// keeping historical positions
// ========Step 1, create scruct=======
currentpos.x := rCurrentX;
currentpos.y := rCurrentY;

// ========Step 2, every 0.5 seconds, set new data to be index 0, and do a SHIFT command to the right=======
timer(IN := TRUE, PT := T#0.5S);
IF timer.Q THEN
	hist[1,0] := currentpos;
	FOR i := len-1 TO 1 BY -1 DO
	  hist[1,i] := hist[1,i-1];
	END_FOR 
	timer(IN := FALSE);
END_IF
// ===========================================================================
// =========Just to get local ams net id for python script========
IF bReqStarted THEN
	fbAms(bExecute := TRUE, tTimeOut := T#2S);
	IF NOT fbAms.bBusy THEN
		fbAms(bExecute := FALSE);
		bReqStarted := FALSE;
	END_IF
END_IF

METHOD Round2dp : REAL
VAR_INPUT
	rNum : REAL;
END_VAR
Round2dp := INT_TO_REAL(REAL_TO_INT(rNum * 100))/100;
END_METHOD

END_PROGRAM

// ---- POUs/MovementType_Teach/FB_Movement_Xbox.TcPOU
FUNCTION_BLOCK FB_Movement_Xbox
VAR_INPUT
	bExecute : BOOL;
	balluff_pos	AT %I* 	: BOOL;
	balluff_neg	at %I* 	: BOOL;
	leftSwitch	at %I* 	: BOOL;
	rightSwitch	at %I* 	: BOOL;
END_VAR
VAR_OUTPUT
END_VAR
VAR
	caseswitch : (init, activatexbox, movement, teachframe, inputarrangement, arrange, map, startmovement, end, errorhandler, error);
	
	// xbox controls
	bXboxUp : BOOL;
	bXboxRight : BOOL;
	bXboxDown : BOOL;
	bXboxLeft : BOOL;
	ProcessXbox : NT_StartProcess;
	
	// HMI controls
	bBtnTeach : BOOL; 
	bBtnArrange : BOOL;
	bBtnConfirmArrangement : BOOL;
	bBtnStartMovement : BOOL;
	BtnTeachTrig : R_TRIG;
	BtnArrangeTrig : R_TRIG;
	BtnConfirmArrangementTrig : R_TRIG;
	BtnStartMovementTrig : R_TRIG;
	
	// Frames to memorise positions
	Frames : FB_Frames;
	// Placeholder to hold current frame name
	sFrameName : STRING;
	msg : STRING; 
	// Frame Arrangement
	sTotalFramesString : STRING(700);
	aFramesString : ARRAY[0..60] OF STRING;
	
	// To split strings into frames
	poop : ARRAY[0..60] OF STRING;
	i : INT;
	bResultSplit : BOOL;
	sSeperator : STRING := '\n';
	iUntitledFrame : INT;
	
	// kinematics FBs
	initPGT : R_TRIG; // used to detect first invokation of FB, stands for initialising postive going transition
	fbMover : FB_HbotMovement;
	fbHome : FB_HbotHome;
	(* 20230711: Added Homing FBs to bypass existing homing method *)
	StepperAHome : MC_Home;
	StepperBHome : MC_Home;
	
	StepperAJog : MC_Jog;
	StepperBJog : MC_Jog;
	joggers : ARRAY[0..1] OF ARRAY[0..1] OF BOOL;
	
	// To Start Movement
	fbTeachMove : FB_Movement_Teach;
	
	//Limit Switches	
	
	LEFTUPPERSENSOR : BOOL;
	LEFTLOWERSENSOR : BOOL;
	RIGHTUPPERSENSOR : BOOL;
	RIGHTLOWERSENSOR : BOOL;
	LEFTTROLLEYSENSOR : BOOL;
	RIGHTTROLLEYSENSOR : BOOL;
	
	(* 20230929: Attempting to use Analog controls for movement - HbotKinematics *)
	hbotCalc : FB_HbotKinematics;
	ABVelo : ARRAY [0..1] OF REAL;
	
	XYVelo: ARRAY [0..1] OF REAL;
	
END_VAR

BtnTeachTrig(CLK := bBtnTeach);
BtnArrangeTrig(CLK := bBtnArrange);
BtnConfirmArrangementTrig(CLK := bBtnConfirmArrangement);
BtnStartMovementTrig(CLK := bBtnStartMovement);
initPGT(CLK := bExecute);

IF balluff_pos THEN //x Maximum reached
	IF TcXbox.xBoxController.P_Left_Joystick.fY > 0 THEN //remember that Y in xbox is x in Frame
		XYVelo[0] := 0;
	ELSE
		XYVelo[0] := TcXbox.xBoxController.P_Left_Joystick.fY;
	END_IF
ELSIF balluff_neg THEN
	IF TcXbox.xBoxController.P_Left_Joystick.fY < 0 THEN //remember that Y in xbox is x in Frame
		XYVelo[0] := 0;
	ELSE 
		XYVelo[0] := TcXbox.xBoxController.P_Left_Joystick.fY;
	END_IF
ELSE
	XYVelo[0] := TcXbox.xBoxController.P_Left_Joystick.fY;
END_IF

IF leftSwitch THEN //x Maximum reached
	IF TcXbox.xBoxController.P_Left_Joystick.fX< 0 THEN //remember that X in xbox is Y in Frame
		XYVelo[1] := 0;
	ELSE
		XYVelo[1] := TcXbox.xBoxController.P_Left_Joystick.fX;
	END_IF
ELSIF RightSwitch THEN
	IF TcXbox.xBoxController.P_Left_Joystick.fX > 0 THEN //remember that X in xbox is Y in Frame
		XYVelo[1] := 0;
	ELSE
		XYVelo[1] := TcXbox.xBoxController.P_Left_Joystick.fX;
	END_IF
ELSE
	XYVelo[1] := TcXbox.xBoxController.P_Left_Joystick.fX;
END_IF

IF initPGT.Q THEN // if the FB just started running, set case to init case to HOME (safety)
	caseswitch := activatexbox;
END_IF

IF bExecute THEN
	
	CASE caseswitch OF 
(*		init:
		(* 20230711: without proper limit switches homing is difficult *)
		(* Homing with Set Position will be done instead *)
		
			(* Existing Homing *)
			fbHome(bExecute := TRUE, StepperA := GVL.StepperReferenceA, StepperB := GVL.StepperReferenceB,
				limitSwitchX := GVL.LimitSwitchX, limitSwitchY := GVL.LimitSwitchY);
			IF fbHome.bError THEN
				caseswitch := error;
			ELSIF fbHome.bDone THEN
				fbHome(bExecute := FALSE, StepperA := GVL.StepperReferenceA, StepperB := GVL.StepperReferenceB,
				limitSwitchX := GVL.LimitSwitchX, limitSwitchY := GVL.LimitSwitchY);
				caseswitch := activatexbox;
			END_IF
			
			(* Current Homing - typically would be manually moving the axis to the centre before pressing Start *)
			//StepperAHome(axis := gvl.StepperReferenceA, execute := TRUE, homingmode := MC_Direct, position := 0);
			//StepperBHome(axis := gvl.StepperReferenceB, execute := TRUE, homingmode := MC_Direct, position := 0);
			//IF stepperaHome.Done AND NOT stepperaHome.CommandAborted AND
			//	
			//	
			//END_IF *)
			
		activatexbox:
			caseswitch := movement;
		
		movement:
		(* 20230711: DPad Buttons don't tally with the actual HBOT Frame, current (correct) config below *)
			(*joggers := RunXboxJogger(Up := TcXbox.xBoxController.P_Buttons.DPad.bRight, Right := TcXbox.xBoxController.P_Buttons.DPad.bUp, Down := TcXbox.xBoxController.P_Buttons.DPad.bLeft, Left := TcXbox.xBoxController.P_Buttons.DPad.bDown);
			StepperAJog(Axis := GVL.StepperReferenceA, JogForward := joggers[0][0], JogBackwards := joggers[0][1], Velocity := 100);
			StepperBJog(Axis := GVL.StepperReferenceB, JogForward := joggers[1][0], JogBackwards := joggers[1][1], Velocity := 100);*)
{'Region' := 'Analog Joystick Movement'}			
		(* 20230929: Attempting to use Analog controls for movement *)
		(*abVelo := hbotCalc.CalculateVelocities(rDeltaX:= TcXbox.xBoxController.P_Left_Joystick.fX, 
												rDeltaY:= TcXbox.xBoxController.P_Left_Joystick.fY, 
												rLinearSpeed:= 100.0);*)
		//oriented 90deg i.e. flip X and Y Axes
		//20231003: 
		(*
			IF LEFTSENSOR OR RIGHTSENSOR THEN
				TcXbox.xBoxController.P_Left_Joystick.fY > 0 then				
					TcXbox.xBoxController.P_Left_Joystick.fY := 0;
		*)
		abVelo := hbotCalc.CalculateAxisRotationRelative(rDeltaX:= (XYVelo[0]*1.6), 
															rDeltaY:= (XYVelo[1])*1.6);
		IF abvelo[0] > 0 THEN
			StepperAJog.JogForward := TRUE;
			StepperAJog.JogBackwards := FALSE;			
		ELSIF abvelo[0] < 0 THEN
			StepperAJog.JogForward := FALSE;
			StepperAJog.JogBackwards := TRUE;
		ELSE
			StepperAJog.JogForward := FALSE;
			stepperAJog.JogBackwards := FALSE;
		END_IF
		IF abvelo[1] > 0 THEN
			StepperbJog.JogForward := TRUE;
			StepperbJog.JogBackwards := FALSE;
		ELSIF abvelo[1] < 0 THEN
			StepperbJog.JogForward := FALSE;
			StepperbJog.JogBackwards := TRUE;
		ELSE
			StepperbJog.JogForward := FALSE;
			stepperbJog.JogBackwards := FALSE;
		END_IF
		//Use MC_JOGMODE_CONTINUOUS so that Velocity actually does something lmao
		StepperAJog(Axis := GVL.StepperReferenceA, Velocity := ABS(abvelo[0]), mode := E_JogMode.MC_JOGMODE_CONTINOUS);
		StepperBJog(Axis := GVL.StepperReferenceB, Velocity := ABS(abvelo[1]), mode := E_JogMode.MC_JOGMODE_CONTINOUS);
{'endregion'}			
		
			IF BtnTeachTrig.Q THEN
				caseswitch := teachframe;
			END_IF
			IF BtnArrangeTrig.Q THEN
				caseswitch := inputarrangement;
			END_IF
			IF BtnStartMovementTrig.Q THEN
				caseswitch := startmovement;
			END_IF
		
		teachframe:
			IF sFrameName = '' THEN
				sFrameName := CONCAT('Unititled', INT_TO_STRING(iUntitledFrame));
				IF (Frames.Teach(sName := sFrameName, rX := HbotForwardKinematics.rCurrentX, rY := HbotForwardKinematics.rCurrentY)) THEN
					iUntitledFrame := iUntitledFrame + 1;
					sFrameName := '';
					caseswitch := movement;
				END_IF
			ELSIF (Frames.Teach(sName := sFrameName, rX := HbotForwardKinematics.rCurrentX, rY := HbotForwardKinematics.rCurrentY)) THEN
				caseswitch := movement;
			END_IF
			
		inputarrangement:
	//		IF BtnConfirmArrangementTrig.Q THEN
				IF sTotalFramesString <> '' THEN
					caseswitch := arrange;
				END_IF
	//		END_IF
			
		arrange:
			// split sTotalFramesString into array of string based on the new line seperator
			MEMSET(ADR(aFramesString), fillByte :=0, n := SIZEOF(aFramesString));
			aFramesString[0] := sTotalFramesString;
			FOR i := 0 TO 59 DO
				bResultSplit := FindAndSplit(	pSeparator := ADR(sSeperator),
												pSrcString := ADR(aFramesString[i]),
												pLeftString := ADR(aFramesString[i]),
												nLeftSize := SIZEOF(aFramesString[i]),
												pRightString := ADR(aFramesString[i+1]),
												nRightSize := SIZEOF(aFramesString[i+1]),
												bSearchFromRight:=FALSE);
				IF NOT bResultSplit THEN
					caseswitch := map;
					EXIT;
				END_IF
			END_FOR
			
		map:
			Frames.Map(aFramesString);
			caseswitch := movement;
			
			
			
		startmovement:
			fbTeachMove(bExecute := TRUE, aArrangedFrames := Frames.ArrangedFrames);
			IF fbTeachMove.bExit THEN
				fbTeachMove(bExecute := FALSE);
				caseswitch := movement;
			END_IF
	END_CASE

END_IF

METHOD RunXboxJogger : ARRAY [0..1] OF ARRAY [0..1] OF BOOL;
VAR_INPUT
	Left : BOOL;
	Right : BOOL;
	Up : BOOL;
	Down : BOOL;
END_VAR
VAR
	StepA : INT;
	StepB : INT;
	bStepAForward : BOOL;
	bStepABackward : BOOL;
	bStepBForward : BOOL;
	bStepBBackward : BOOL;
	placeHolder : ARRAY [0..1] OF ARRAY [0..1] OF BOOL;
END_VAR
IF Left THEN
	StepA := StepA + 1;
	StepB := StepB + 1;
END_IF

IF Down THEN
	StepA := StepA + 1;
	StepB := StepB - 1;
END_IF

IF Right THEN
	StepA := StepA - 1;
	StepB := StepB - 1;
END_IF

IF Up THEN
	StepA := StepA - 1;
	StepB := StepB + 1;
END_IF

IF StepA > 0 THEN
	placeHolder[0][0] := TRUE;
ELSIF StepA < 0 THEN
	placeHolder[0][1] := TRUE;
END_IF

IF StepB > 0 THEN
	placeHolder[1][0] := TRUE;
ELSIF StepB < 0 THEN
	placeHolder[1][1] := TRUE;
END_IF
RunXboxJogger := placeHolder;
END_METHOD

END_FUNCTION_BLOCK

// ---- POUs/MovementType_Teach/FB_Frames.TcPOU
FUNCTION_BLOCK FB_Frames
VAR_INPUT
END_VAR
VAR_OUTPUT
END_VAR
VAR
	AllFrames : ARRAY[0..40] OF Frame;
	ArrangedFrames : ARRAY[0..60] OF Frame;
	i: INT;
END_VAR

METHOD Map : ARRAY[0..60] OF Frame
VAR_INPUT
	aFrameString : ARRAY[0..60] OF STRING;
END_VAR
VAR
	i : INT;
	j : INT;
	PlaceHolder : ARRAY[0..60] OF Frame;
END_VAR
FOR i := 0 TO 60 DO
	IF aFrameString[i] = '' THEN
		PlaceHolder[i].Name := ''; 
		PlaceHolder[i].X := 0; 
		PlaceHolder[i].Y := 0; 
	ELSE
		FOR j := 0 TO 60 DO
			IF aFrameString[i] = AllFrames[j].Name THEN
				PlaceHolder[i] := AllFrames[j];
			ELSIF AllFrames[j].Name = '' THEN
				EXIT;
			END_IF
		END_FOR
		j := 0;
	END_IF
END_FOR
ArrangedFrames := PlaceHolder;
Map := PlaceHolder;
END_METHOD

METHOD Teach : BOOL
VAR_INPUT
	sName : STRING;
	rX : REAL;
	rY : REAL;
END_VAR
VAR
	i : INT;
END_VAR
FOR i := 0 TO 30 BY 1 DO
	IF AllFrames[i].Name = '' AND AllFrames[i].X = 0 AND AllFrames[i].Y = 0 THEN
		AllFrames[i].Name := sName;
		AllFrames[i].X := rX;
		AllFrames[i].Y := rY;
		Teach := TRUE;
		EXIT;
	END_IF
END_FOR
END_METHOD

END_FUNCTION_BLOCK

// ---- POUs/MovementType_Teach/FB_Movement_Teach.TcPOU
FUNCTION_BLOCK FB_Movement_Teach
VAR_INPUT
	bExecute : BOOL;
	aArrangedFrames : ARRAY[0..60] OF Frame;
END_VAR
VAR_OUTPUT
END_VAR
VAR
	caseswitch : (init, prepare, executemovement, end, error);
	
	initPGT : R_TRIG; // used to detect first invokation of FB, stands for initialising postive going transition
	fbMover : FB_HbotMovement;
	fbHome : FB_HbotHome;
	iFrameCount : INT := 0;
	bNextFrame : BOOL;
	
	// HMI controls
	bRunSequence : BOOL;
	bRepeat : BOOL;
	bAbort : BOOL;
	bEnableHmiButton : BOOL; // This is to enable the HMI Buttons like abort, run sequence, repear...
	bExit: BOOL;
END_VAR

initPGT(CLK := bExecute);
IF initPGT.Q THEN // if the FB just started running, set case to init case to HOME (safety)
	iFrameCount := 0;
	caseswitch := prepare;
	bAbort := FALSE;
	bExit := FALSE;
	bEnableHmiButton := TRUE;
END_IF

CASE caseswitch OF 
//	init:
//		fbHome(bExecute := TRUE, StepperA := GVL.StepperReferenceA, StepperB := GVL.StepperReferenceB,
//			limitSwitchX := GVL.LimitSwitchX, limitSwitchY := GVL.LimitSwitchY);
//		IF fbHome.bError THEN
//			caseswitch := error;
//		ELSIF fbHome.bDone THEN
//			fbHome(bExecute := FALSE, StepperA := GVL.StepperReferenceA, StepperB := GVL.StepperReferenceB,
//			limitSwitchX := GVL.LimitSwitchX, limitSwitchY := GVL.LimitSwitchY);
//			caseswitch := prepare;
//		END_IF
		
	prepare:
		fbMover( bExecute := FALSE, StepperA := GVL.StepperReferenceA, StepperB := GVL.StepperReferenceB); // stop all movement
		IF aArrangedFrames[iFrameCount].Name = '' THEN
			iFrameCount := 0;
			
		END_IF
		
		IF bAbort THEN
			bExit := TRUE;	
			bEnableHmiButton := FALSE;
		ELSIF NOT bAbort THEN		
			IF bRunSequence THEN
				IF iFrameCount = 0 AND NOT bNextFrame THEN
					caseswitch := executemovement;
				ELSE
					iFrameCount := iFrameCount + 1;
					caseswitch := executemovement;
				END_IF
			END_IF
		END_IF
		
	executemovement:
		fbMover(MovementMode := fbMover.MoveAbsolute,
				rLinearSpeed := 60,
				rCurrentX := HbotForwardKinematics.rCurrentX,
				rCurrentY := HbotForwardKinematics.rCurrentY,
				rDeltaX := aArrangedFrames[iFrameCount].X,
				rDeltaY := aArrangedFrames[iFrameCount].Y,
				bExecute := TRUE,
				StepperA := GVL.StepperReferenceA,
				StepperB := GVL.StepperReferenceB);
		IF fbMover.bError THEN
			caseswitch := error; //catch errors
		ELSIF fbMover.bDone THEN
			bNextFrame := TRUE;
			caseswitch := prepare; // if it is done, go to the prep switch case
		END_IF
		IF NOT bRepeat THEN
			bRunSequence := FALSE;
		END_IF
		
END_CASE

END_FUNCTION_BLOCK

// ---- POUs/E_Stop.TcPOU
PROGRAM E_Stop
VAR
	estoprtrig : R_TRIG ;
	Resetrtrig : R_TRig;
	
	UserResetButton AT %I*: BOOL; 			(* Input signal for manual Reset activation *) // LINK TO GVL.ResetButton
	UserEStopButton AT %I*: BOOL ; 			(* Input signal for manual E-stop activation *) // LINK TO GVL.EstopButton
    EStop : BOOL := FALSE;				(* Emergency stop internal flag *)
	
	StopMotorA : MC_Stop;
	StopMotorB : MC_Stop;
	ResetMotorA : MC_Reset;
	ResetMotorB : MC_Reset;
	
	casestate : INT;
END_VAR

CASE  casestate  OF 
	0 : //initialisation.
		casestate := 10;
		
	10 : // Check If E_Stop isTriggered 
	IF  UserEStopButton = FALSE THEN 
		 StopMotorA(Execute := TRUE, Axis:= GVL.StepperReferenceA) ;  (* actual function to stop the motor *)
		 StopMotorB(Execute := TRUE,Axis:= GVL.StepperReferenceB) ;  (* actual function to stop the motor *)
		 casestate := 20; 
		 ELSE 
		ResetMotorA (Execute := FALSE, Axis := GVL.StepperReferenceA); (*Reset the Motors *)
		ResetMotorB (Execute := FALSE, Axis := GVL.StepperReferenceB); (*Reset the Motors *)
			 //chill again. Wait for Lim Switch Activation 
	END_IF
	
	20 : // Wait for Limit Switches to NOT be pressed before allowing movement again
	IF UserResetButton THEN
		casestate := 30 ;
		ELSE 
			//chill	
	END_IF
			
	30 : 
		
		IF StopMotorA.Active = FALSE THEN // IF FB not active, stop and start the FB 
		StopMotorA(Execute := TRUE, Axis:= GVL.StepperReferenceA) ;  (* actual function to stop the motor *)
		StopMotorB(Execute := TRUE,Axis:= GVL.StepperReferenceB) ;  (* actual function to stop 

the motor *)
		casestate := 40; 
		ELSIF StopMotorA.Active = TRUE THEN  //After Stopping and Starting, If ACtive = True continue as per normal
		ResetMotorA (Execute := TRUE, Axis := GVL.StepperReferenceA); (*Reset the Motors *)
		ResetMotorB (Execute := TRUE, Axis := GVL.StepperReferenceB); (*Reset the Motors *)
		StopMotorA(Execute := FALSE, Axis:= GVL.StepperReferenceA) ;  (* actual function to continue the motor *)
		StopMotorB(Execute := FALSE,Axis:= GVL.StepperReferenceB) ;  (* actual function to continue the motor *)
		casestate := 0;
		END_IF
	40 :  // Buffer for resetting the FB 
		casestate := 30;
		
END_CASE

END_PROGRAM

// ---- POUs/LimitSwitches.TcPOU
PROGRAM LimitSwitches
VAR
	StopMotorA : MC_Stop;
	StopMotorB : MC_Stop;
	ResetMotorA : MC_Reset;
	ResetMotorB : MC_Reset;
	
	casestate : INT;
END_VAR

CASE  casestate  OF 
	0 : //initialisation. If Axis is ready, then prepare to hit limit switch, if not, do nothing
	IF  PrepareAxes.switchcase = Implicit_Enum__PrepareAxes__switchcase.Movement THEN 
		casestate := 10;
		ELSE 
			//chill here
	END_IF
	10 : // Check If Limit Switch Triggered 
	IF GVL.LimitSwitchBotLeft OR GVL.LimitSwitchBotRight OR GVL.LimitSwitchMidLeft OR GVL.LimitSwitchMidRight OR GVL.LimitSwitchTopLeft OR GVL.LimitSwitchTopRight THEN 
		 StopMotorA(Execute := TRUE, Axis:= GVL.StepperReferenceA) ;  (* actual function to stop the motor *)
		 StopMotorB(Execute := TRUE,Axis:= GVL.StepperReferenceB) ;  (* actual function to stop the motor *)
		 casestate := 20; 
		 ELSE 
		ResetMotorA (Execute := FALSE, Axis := GVL.StepperReferenceA); (*Reset the Motors *)
		ResetMotorB (Execute := FALSE, Axis := GVL.StepperReferenceB); (*Reset the Motors *)
			 //chill again. Wait for Lim Switch Activation 
	END_IF
	
	20 : // Wait for Limit Switches to NOT be pressed before allowing movement again
	IF GVL.LimitSwitchBotLeft = FALSE AND GVL.LimitSwitchBotRight = FALSE AND GVL.LimitSwitchMidLeft = FALSE AND GVL.LimitSwitchMidRight = FALSE AND GVL.LimitSwitchTopLeft = FALSE AND GVL.LimitSwitchTopRight = FALSE THEN 
		casestate := 30 ;
		ELSE 
			//chill	
	END_IF
			
	30 : 
		
		IF StopMotorA.Active = FALSE THEN // IF FB not active, stop and start the FB 
		StopMotorA(Execute := TRUE, Axis:= GVL.StepperReferenceA) ;  (* actual function to stop the motor *)
		StopMotorB(Execute := TRUE,Axis:= GVL.StepperReferenceB) ;  (* actual function to stop the motor *)
		casestate := 40; 
		ELSIF StopMotorA.Active = TRUE THEN  //After Stopping and Starting, If ACtive = True continue as per normal
		ResetMotorA (Execute := TRUE, Axis := GVL.StepperReferenceA); (*Reset the Motors *)
		ResetMotorB (Execute := TRUE, Axis := GVL.StepperReferenceB); (*Reset the Motors *)
		StopMotorA(Execute := FALSE, Axis:= GVL.StepperReferenceA) ;  (* actual function to continue the motor *)
		StopMotorB(Execute := FALSE,Axis:= GVL.StepperReferenceB) ;  (* actual function to continue the motor *)
		casestate := 0;
		END_IF
	40 :  // Buffer for resetting the FB 
		casestate := 30;
		
END_CASE

END_PROGRAM
